(* CODESYS project Domains.library
   Company: _
   DefaultNamespace: Domains
   Title: Domains
   Placeholder: _Domains
   Author: Krystian Lis et al.
   Description: Each Domain should have a number of standard browsable components.
   Version: 1.0.0

Project tree, tasks and I/O mapping:
  libraries: Debug, * (_); Results, * (_); Tc2_Standard, * (Beckhoff Automation GmbH); Tc3_Module, * (Beckhoff Automation GmbH); Calls, * (_)
  Domain/
    _/
      global variables _Register
      function _RegisterDomain [ST]
      interface I_DomainInternal: CTable, IsRegistered
      global variables Param
    Component/
      function block CTable [ST]: Cap, Get, Insert, Length
      interface I_Component
      interface I_CTable: Cap, Get, Length
      interface I_MutCTable: Insert
    Domain/
      function block Domain [ST]: CTable, FB_init, IsRegistered, Self
      function GetDomain [ST]
      interface I_Domain: CTable
      interface I_DomainProvider: Self
*)

// Domain/_/_Register
{attribute 'qualified_only'}
VAR_GLOBAL INTERNAL
	iDomain			: ARRAY[1..Param.MAX_DOMAIN] OF I_DomainInternal;
	nLen			: UDINT := 0;
END_VAR

// Domain/_/Param
{attribute 'qualified_only'}
VAR_GLOBAL CONSTANT
	MAX_DOMAIN : UDINT := 100;
END_VAR

// Domain/_/_RegisterDomain
FUNCTION INTERNAL _RegisterDomain : Results.Result
VAR_INPUT
	iDomain			: I_DomainInternal;
END_VAR

IF iDomain = 0 THEN
	Debug.DebugMsg(0, Tc2_Standard.CONCAT(__POUNAME(), 'iDomain = 0!'));
	_RegisterDomain := Results.Err.Itf0;
	RETURN;
END_IF

IF iDomain.IsRegistered THEN
	Debug.DebugMsg(iDomain, Tc2_Standard.CONCAT(__POUNAME(), 'iDomain is already registered!'));
	_RegisterDomain := Results.Err.Itf0;
	RETURN;
END_IF

IF _Register.nLen = Param.MAX_DOMAIN THEN
	Debug.DebugMsg(iDomain, Tc2_Standard.CONCAT(__POUNAME(), 'Overflow!'));
	_RegisterDomain := Results.Err.Ovf;
	RETURN;
END_IF

_Register.nLen := _Register.nLen + 1;
_Register.iDomain[_Register.nLen] := iDomain;
_RegisterDomain := Results.Ok;

END_FUNCTION

// Domain/_/I_DomainInternal
INTERFACE INTERNAL I_DomainInternal EXTENDS I_Domain

PROPERTY CTable : I_CTable
GET
END_GET
END_PROPERTY

PROPERTY INTERNAL IsRegistered : BOOL
GET
END_GET
SET
END_SET
END_PROPERTY

END_INTERFACE

// Domain/Domain/I_Domain
INTERFACE I_Domain EXTENDS Debug.I_Debug;

PROPERTY CTable : I_CTable
GET
END_GET
END_PROPERTY

END_INTERFACE

// Domain/Component/CTable
FUNCTION_BLOCK CTable
VAR_GENERIC CONSTANT
	nMaxIndex	: UDINT := 100;
END_VAR

IMPLEMENTS I_CTable

VAR
	_iTable	: ARRAY[1..nMaxIndex] OF I_Component;
	_nLen	: UDINT := 0;
END_VAR

PROPERTY Cap : UDINT
GET
Cap := nMaxIndex;
END_GET
END_PROPERTY

METHOD Get : Results.Result
VAR_INPUT
	nIndex		: UDINT;
END_VAR
VAR_OUTPUT
	iComponent	: I_Component;
END_VAR
IF _nLen = 0 THEN
	RETURN;
END_IF

IF nIndex > _nLen THEN
	RETURN;
END_IF

IF nIndex > nMaxIndex OR_ELSE nIndex < 1 THEN
	Get := Results.Err.Ovf;
	RETURN;
END_IF

iComponent := _iTable[nIndex];
Get := Results.Ok;
END_METHOD

METHOD Insert : Results.Result
VAR_INPUT
	iComponent	: I_Component;
END_VAR
VAR_OUTPUT
	nIndex		: UDINT;
END_VAR
VAR
	i			: UDINT;
END_VAR
IF iComponent = 0 THEN
	Insert := Results.Err.Itf0;
	RETURN;
END_IF

IF _nLen = nMaxIndex THEN
	Insert := Results.Err.Ovf;
	RETURN;
END_IF

FOR i := 1 TO nMaxIndex DO
	IF _iTable[i] = iComponent THEN		
		Insert := Results.Err.ItfEq;
		RETURN;	
	END_IF
END_FOR

_nLen := _nLen + 1;
_iTable[_nLen] := iComponent;
Insert := Results.Ok;
END_METHOD

PROPERTY Length : UDINT
GET
Length := _nLen;
END_GET
END_PROPERTY

END_FUNCTION_BLOCK

// Domain/Component/I_CTable
INTERFACE I_CTable EXTENDS Debug.I_Debug

PROPERTY Cap : UDINT
GET
END_GET
END_PROPERTY

METHOD Get : Results.Result
VAR_INPUT
	nIndex		: UDINT;
END_VAR
VAR_OUTPUT
	iComponent	: I_Component;
END_VAR
END_METHOD

PROPERTY Length : UDINT
GET
END_GET
END_PROPERTY

END_INTERFACE

// Domain/Component/I_Component
INTERFACE I_Component EXTENDS Calls.I_Arg

END_INTERFACE

// Domain/Component/I_MutCTable
INTERFACE I_MutCTable EXTENDS I_CTable

METHOD Insert : Results.Result
VAR_INPUT
	iComponent	: I_Component;
END_VAR
VAR_OUTPUT
	nIndex		: UDINT;
END_VAR
END_METHOD

END_INTERFACE

// Domain/Domain/Domain
FUNCTION_BLOCK Domain IMPLEMENTS I_Domain, I_DomainProvider, I_DomainInternal
VAR
	_iCTable		: I_CTable;
	_bIsRegistered	: BOOL;
END_VAR

PROPERTY CTable : I_CTable
GET
CTable := _iCTable;
END_GET
END_PROPERTY

//FB_Init is always available implicitly and it is used primarily for initialization.
//The return value is not evaluated. For a specific influence, you can also declare the
//methods explicitly and provide additional code there with the standard initialization
//code. You can evaluate the return value.
METHOD FB_Init: BOOL
VAR_INPUT
    bInitRetains: BOOL; // TRUE: the retain variables are initialized (reset warm / reset cold)
    bInCopyCode: BOOL;  // TRUE: the instance will be copied to the copy code afterward (online change)
	
	iCTable		: I_CTable;
END_VAR
IF iCTable <> 0 THEN
	_iCTable := iCTable;
	_RegisterDomain(THIS^);
ELSE
	Debug.DebugMsg(THIS^, 'iCTable = 0!');
END_IF
END_METHOD

PROPERTY INTERNAL IsRegistered : BOOL
GET
IsRegistered := _bIsRegistered;
END_GET
SET
_bIsRegistered := IsRegistered;
END_SET
END_PROPERTY

PROPERTY Self : I_Domain
GET
Self := THIS^;
END_GET
END_PROPERTY

END_FUNCTION_BLOCK

// Domain/Domain/I_DomainProvider
INTERFACE I_DomainProvider EXTENDS I_Component

PROPERTY Self : I_Domain
GET
END_GET
END_PROPERTY

END_INTERFACE

// Domain/Domain/GetDomain
FUNCTION GetDomain : Results.Result
VAR_INPUT
	nIndex		: UDINT := 0;
END_VAR
VAR_OUTPUT
	iDomain		: I_Domain;
END_VAR

IF nIndex >= _Register.nLen THEN
	GetDomain := Results.None;
	RETURN;
END_IF

iDomain := _Register.iDomain[nIndex];
IF iDomain <> 0 THEN
	GetDomain := Results.Ok;
	RETURN;
END_IF

END_FUNCTION
